% RSLogix 500 project P5.RSS, saved by version 12.00.00.00 %
PROJECT "UNTITLED"    % processor: Bul.1763 MicroLogix 1100 Series B %

PROGRAM FILES
  LAD 2   5 rungs

DATA FILES
  O0 OUTPUT  4 elements
  I1 INPUT  6 elements
  S2 STATUS  66 elements
  B3 BINARY  1 elements
  T4 TIMER  1 elements
  C5 COUNTER  1 elements
  R6 CONTROL  1 elements
  N7 INTEGER  1 elements
  F8 FLOAT  2 elements

LADDER 2
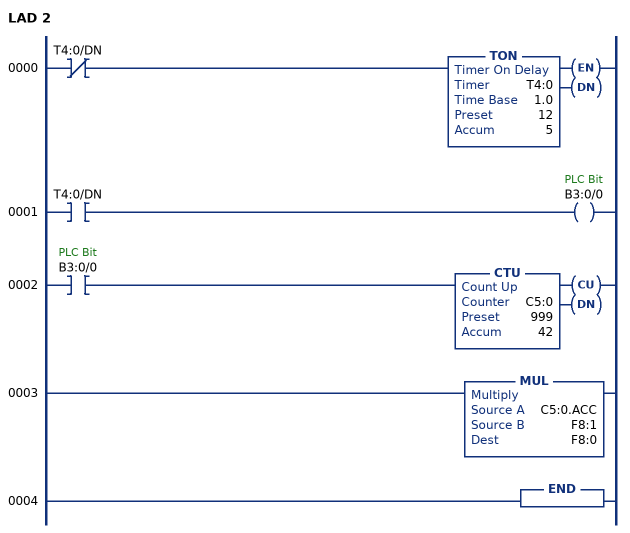
% Rung: 0 %
SOR XIO T4:0/DN TON T4:0 1.0 12 5 EOR
% Rung: 1 %
SOR XIC T4:0/DN OTE B3:0/0 EOR
%   B3:0/0  "PLC Bit" %
% Rung: 2 %
SOR XIC B3:0/0 CTU C5:0 999 42 EOR
%   B3:0/0  "PLC Bit" %
% Rung: 3 %
SOR MUL C5:0.ACC F8:1 F8:0 EOR
% Rung: 4 %
SOR END EOR

DATA TABLE (non-zero values as saved)
DATA T4
% .PRE .ACC %
% T4:0 % 12 5
DATA C5
% .PRE .ACC %
% C5:0 % 999 42
DATA F8
% F8:0 % 256.2 6.1
